{attribute 'qualified_only'}
VAR_GLOBAL
END_VAR

(* stored: Version 1.1.0.1
   GVL MAIN_VISION_COMM_VARS: Id {27e6601a-46e6-42c7-8d84-79ba14347407} *)
